Staubli VAL3: page_trajectory.pjx

--- page_trajectory.pjx ---
Parameters version=s7.8.3 stackSize=5000 millimeterUnit=true
Program file=alreadyExist.pgx
Program file=buildList.pgx
Program file=cleanUserMenu.pgx
Program file=defineTraj.pgx
Program file=deleteItem.pgx
Program file=goTo.pgx
Program file=listAdd.pgx
Program file=loadPage.pgx
Program file=main.pgx
Program file=onEnterEvent.pgx
Program file=onExit.pgx
Program file=onF1Event.pgx
Program file=onF2Event.pgx
Program file=onF3Event.pgx
Program file=onF4Event.pgx
Program file=onF5Event.pgx
Program file=onF6Event.pgx
Program file=onF7Event.pgx
Program file=onF8Event.pgx
Program file=onLeftEvent.pgx
Program file=onRightEvent.pgx
Program file=onStart.pgx
Program file=refresh.pgx
Program file=refreshDynamic.pgx
Program file=refreshStatic.pgx
Program file=selectType.pgx
Program file=showStatus.pgx
Data file=page_trajectory.dtx
Library alias=use path=Disk://public_temp/userPage/userPage.pjx
Library alias=pub path=Disk://public_temp/pub/pub.pjx
Library alias=data path=Disk://SaveData/SaveData.pjx
Library alias=cycle path=Disk://cycle/cycle.pjx

--- page_trajectory.dtx ---
num nIndex
num nKey = -1
public num nPage
num nRefresh = 2164.601
num nSelected
num nTime = 0.1
num nView
num nType
string sEvent = "hello"
string sEventImport
string sImport
public string sItems
string sList = "hello"
string sMenu[8]
  [0] = "Simulation"
  [4] = "Type"
  [5] = "Duplicate"
  [6] = "Delete"
  [7] = "New"
string sMenu8[8]
string sMenuUser[8]
string sMessage
bool bButton[8]
  [4] = true
  [5] = true
  [6] = true
  [7] = true
bool bLarge
num nIndexItem
num nOldIndex
bool bTrigger
num nClockStatus
bool bShowStatus
bool bMoveRelease
string sWorkingmode[8]
  [0] = "0 安全过度点 Joint"
  [1] = "1 Appro"
pointRx pPointTest[7]
  [0] = {fatherId=world[0]}
  [1] = {fatherId=world[0]}
  [2] = {fatherId=world[0]}
  [3] = {fatherId=world[0]}
  [4] = {fatherId=world[0]}
  [5] = {fatherId=world[0]}
  [6] = {fatherId=world[0]}
string sTrsfNum[8 6]

--- main.pgx ---
public program main()
  local bool l_bSave
  local bool l_bOverRide
  local bool l_bOk
  local bool l_bUnreached
  local string l_sMessage
begin
  //  // INIT
    call onStart()
  //  // LOOP UNTIL nKey=255
  //  nIndexItem=0
  do
    call refresh()
    nKey=getKey()
    call use:listevent(nKey,nIndex,sEvent)
    nView=use:nView
    nSelected=nIndex
		data:nPage_Traj=nIndex
    switch nKey
      case 259
        // TAB
        bLarge=!bLarge
      //  call use:setView()
      break
      case 263
        // backSpace rename
        //call onBackEvent(l_bSave)
      break
      case 32
        // space to edit Action
        //call onSpaceEvent()
      break
      case 271
        call onF1Event()
      break
      case 272
        //
        call onF2Event()
      break
      case 273
        //
        call onF3Event()
      break
      case 274
        //
        call onF4Event()
      break
      case 275
        //
        call onF5Event()
      break
      //
      case 276
        call onF6Event()
      break
      case 277
        //
        call onF7Event()
      break
      case 278
        //
        call onF8Event()
      break
      case 270
        //
        call onEnterEvent()
      break
    endSwitch
    //    endIf
    //    l_bOverRide=false
    //    // release the resource
        delay(0)
    //    if nKey==255 and isKeyPressed(289)==true
    //      call language:message(l_sMessage,143)
    //      call use:timerDialog(l_sMessage,3)
    //    endIf
    if workingMode()!=1
      call use:timerDialog("请切换成手动模式",0)
      wait(workingMode()==1)
    endIf
  until nKey==255 and isKeyPressed(289)==false
  use:bUseRefresh=true
  //  // exit
  //  call onExit(l_bSave)
end

--- alreadyExist.pgx ---
program alreadyExist(string& x_sName[], bool& x_bUndo[])
  local num l_nX
  local num l_nY
  local string l_sString
begin
//  // look if the trajectory already exist
//  l_nX=40-use:nBottomX-1
//  l_nY=use:nBottomY+1
//  call language:message(l_sString,21)
//  call use:type(l_nX,l_nY,l_sString)
//  // read the new trajectory
//  call use:read(l_nX+len(l_sString),l_nY,x_sName,10,false)
//  if !use:bUseEscape
//    call trajType:find(x_sName,x_bUndo)
//    if x_bUndo
//      call language:message(x_sName,-2)
//      popUpMsg(x_sName)
//    endIf
//  else
//    x_bUndo=true
//  endIf
end

--- buildList.pgx ---
program buildList()
  local num l_nSize
  local string l_sEvent
  local num i
  local bool l_bFound
  local num l_nCount
  local string l_sEmpty
  local num j
begin
  call use:setSizeList(0,0,38,10)
  //call use:setSizeList(15,0,18,9)
  //建立对话款
  call use:listcreate("第1槽/6槽")
  //  for i=0 to 7
  //    call use:listadd(sMenu[i])
  //  endFor
 //   call use:selectNewField(nSelected,nIndex,nView)
  for i=0 to 7
    sTrsfNum[i,0]=toString("",data:pPoinTest[i].trsf.x)
    sTrsfNum[i,1]=toString("",data:pPoinTest[i].trsf.y)
    sTrsfNum[i,2]=toString("",data:pPoinTest[i].trsf.z)
    sTrsfNum[i,3]=toString("",data:pPoinTest[i].trsf.rx)
    sTrsfNum[i,4]=toString("",data:pPoinTest[i].trsf.ry)
    sTrsfNum[i,5]=toString("",data:pPoinTest[i].trsf.rz)
  endFor

  sWorkingmode[0]="0 安全过度点 Joint"
  sWorkingmode[1]="1 Appro(摆正点，{"+sTrsfNum[1,0]+","+sTrsfNum[1,1]+","+sTrsfNum[1,2]+","+sTrsfNum[1,3]+","+sTrsfNum[1,4]+","+sTrsfNum[1,5]+"})"
  sWorkingmode[2]="2 Appro(摆正点，{"+sTrsfNum[2,0]+","+sTrsfNum[2,1]+","+sTrsfNum[2,2]+","+sTrsfNum[2,3]+","+sTrsfNum[2,4]+","+sTrsfNum[2,5]+"})"
  sWorkingmode[3]="3 Appro(到位点，{"+sTrsfNum[3,0]+","+sTrsfNum[3,1]+","+sTrsfNum[3,2]+","+sTrsfNum[3,3]+","+sTrsfNum[3,4]+","+sTrsfNum[3,5]+"})"
  sWorkingmode[4]="4 Appro(到位点，{"+sTrsfNum[4,0]+","+sTrsfNum[4,1]+","+sTrsfNum[4,2]+","+sTrsfNum[4,3]+","+sTrsfNum[4,4]+","+sTrsfNum[4,5]+"})"
  sWorkingmode[5]="5 Appro(到位点，{"+sTrsfNum[5,0]+","+sTrsfNum[5,1]+","+sTrsfNum[5,2]+","+sTrsfNum[5,3]+","+sTrsfNum[5,4]+","+sTrsfNum[5,5]+"})"
  sWorkingmode[6]="6 Appro(摆正点，{"+sTrsfNum[6,0]+","+sTrsfNum[6,1]+","+sTrsfNum[6,2]+","+sTrsfNum[6,3]+","+sTrsfNum[6,4]+","+sTrsfNum[6,5]+"})"
  sWorkingmode[7]="7 Appro(摆正点，{"+sTrsfNum[7,0]+","+sTrsfNum[7,1]+","+sTrsfNum[7,2]+","+sTrsfNum[7,3]+","+sTrsfNum[7,4]+","+sTrsfNum[7,5]+"})"

  call use:listadd(sWorkingmode)
  call use:selectNewField(nSelected,nIndex,nView)
  call use:listupdate(0)
 // nIndex=data:nPage_Traj
 // call use:selectNewField(nSelected,nIndex,nView)
end

--- cleanUserMenu.pgx ---
program cleanUserMenu()
  local num i
begin
//  // clean all the reference
//  for i=0 to size(sMenuUser)-1
//    sMenuUser[i]=""
//  endFor
end

--- defineTraj.pgx ---
program defineTraj()
  local num i
  local num l_nType
  local string l_sPath
begin
//  // select the trajectory type
//  if saveData:sTrajTypeUsing==""
//    saveData:sTrajTypeUsing=saveData:sTrajType
//  endIf
//  // search inside all the instruction
//  call saveData:getPathInstr(saveData:sTrajTypeUsing,l_sPath)
//  // check the trajType
//  if trajType:libPath()!=l_sPath and l_sPath!=""
//    i=trajType:libLoad(l_sPath)
//    delay(0)
//  endIf
//  // error
//  if i!=0
//    popUpMsg("error load traj type on ENTER"+saveData:sTrajTypeUsing+toString("",i))
//  endIf
end

--- deleteItem.pgx ---
program deleteItem(bool& x_bResult)
  local string l_sSwap
  local num l_nResult
  local string l_sMessage
  local string l_sMessage2
  local bool l_bYes
  local string l_sButton[2]
begin
//  //
//  // delete a Trajectory
//  //
//  x_bResult=false
//  // check
//  if sEvent!=""
//    l_iSwap.sType=saveData:sTrajTypeUsing
//    l_iSwap.sData=sEvent
//    call prog:findItem(l_iSwap,l_nResult,false)
//    if l_nResult==0
//      //delete it
//      call language:message(l_sMessage,81)
//      call language:getYesNo(l_sButton)
//      // ask the yes_no question
//      call use:yes_no(l_sMessage+"#"+saveData:sTrajTypeUsing+" "+sEvent,l_sButton,l_bYes)
//      x_bResult=l_bYes
//    endIf
//  endIf
end

--- goTo.pgx ---
program goTo(num x_nIndex, bool& x_bUnreached[])
  local bool l_bUnreached
  local num l_nIndexTool
  local tool l_tTool
  local num l_nSize
  local string l_sItems[2]
  local num l_nId
  local num l_nResult
begin
//  // check the cycle status
//  if !cycleStatus:bCycle and !cycleStatus:bSimulation
//    // check the working Mode
//    if cycleStatus:nWorkingMode==1 and isPowered()
//      // set the memory for the moveHold button
//      if cycleStatus:nWorkingStatus==6
//        bMoveRelease=true
//      endIf
//      // check for the index
//      if nOldIndex!=x_nIndex or (cycleStatus:nWorkingStatus!=0 and cycleStatus:nWorkingStatus!=6)
//        if !isEmpty()
//          resetMotion()
//        endIf
//        if nOldIndex!=x_nIndex
//          nOldIndex=x_nIndex
//        endIf
//      else
//        if isEmpty() and cycleStatus:nWorkingStatus==0 and bMoveRelease
//          bMoveRelease=false
//          cls()
//          // copy the item to the trajectory
//          l_sItems[0]=sEvent
//          // take the elements
//          call trajType:load(l_sItems,l_nResult)
//          call trajType:getSizeItem(false,l_nSize)
//          // MOVE
//          do
//            if x_nIndex>0
//              call use:typeMenu(7,"<<")
//            else
//              call use:typeMenu(7,"    ")
//            endIf
//            if x_nIndex<=l_nSize
//              call use:typeMenu(8,">>")
//            else
//              call use:typeMenu(8,"    ")
//            endIf
//            // get the data to move
//            call trajType:getTool(l_nIndexTool)
//            call tcp:getTool(l_tTool,l_nIndexTool)
//            call trajType:getTrajItem(l_tTraj,x_nIndex)
//            //
//            // use a sTemp mdesc to set the blend off
//            //
//            l_tTraj.nom_speed.blend=off
//            call trajType:goTo(l_tTool,l_tTraj.nom_speed,l_tTraj.moveType,x_bUnreached,x_nIndex)
//            // TO DO language
//            call use:timerDialog("Going to point: "+toString("",x_nIndex+1)+ " / "+toString("",l_nSize),0)
//            do
//              nKey=getKey()
//              call use:scroll(0,7,38,(getMoveId()-roundDown(getMoveId()))*100)
//              delay(0)
//            until isEmpty()or nKey==255 or nKey==277 or nKey==278
//            // continue
//            if isEmpty() or (nKey==278 and x_nIndex<l_nSize)
//              if isEmpty()
//                call use:timerDialog("At point: "+toString("",x_nIndex+1)+ " / "+toString("",l_nSize),1)
//              endIf
//              x_nIndex=x_nIndex+1
//            elseIf nKey==277 and x_nIndex>0
//              // decrease
//              x_nIndex=x_nIndex-1
//            else
//              delay(1)
//            endIf
//            // release
//            resetMotion()
//          until x_bUnreached or nKey==255 or x_nIndex>=l_nSize or(x_nIndex==l_nSize and l_nSize==1)
//          // refresh
//          use:bUseRefresh=true
//        endIf
//      endIf
//    else
//      // reset the cycle
//      if cycleStatus:nWorkingMode!=1 or !isPowered()
//        resetMotion()
//      endIf
//    endIf
//  endIf
end

--- loadPage.pgx ---
program loadPage(string x_sPage, string& x_sItems[])
// load the next page
  local num i
  local string l_sMessage
begin
//  // look if the page libload is correct
//  i=page:libLoad(x_sPage)
//  delay(0)
//  if i!=0
//    logMsg("[KERNEL] INTERFACE:PAGE LIBLOAD "+x_sPage+" result "+toString("",i))
//    call language:message(l_sMessage,-7)
//    popUpMsg(l_sMessage+x_sPage+" ; "+toString("",i))
//  else
//    // copy all the field from x_sItems to the next page
//    call use:stringCopy(x_sItems,page:sItems)
//    call page:main()
//  endIf
end

--- onExit.pgx ---
program onExit(bool x_bSave)
  local string l_sEmpty
  local num l_nResult
  local string l_sMessage
begin
//  // resetMotion
//  if !cycleStatus:bCycle
//    resetMotion()
//  endIf
//  if x_bSave
//    l_sEmpty=""
//    l_nResult=0
//    call trajType:onSave(l_sEmpty)
//    // show the message
//    call language:message(l_sMessage,-4)
//    call use:timerDialog(l_sMessage,1)
//  endIf
end

--- onF1Event.pgx ---
program onF1Event()
  local bool l_bYes
  local string l_sMessage
  local string l_sItem
  local num l_nResult
begin
//  // look if the bButton is enable
//  if bButton[0]
//    //
//    //SIMULATION
//    //
//    if !cycleStatus:bCycle and sEvent!=""
//      // load the production page
//      call loadPage("Disk://trajectory/page_simulation",sEvent)
//      // save the moveHold
//      bMoveRelease=false
//    endIf
//  endIf
end

--- onF2Event.pgx ---
program onF2Event()
  local string l_sMessage
  local string l_sEvent
  local string l_sFilter
  local num l_nIndex
  local num i
begin
//  // look if the bButton is enable
//  if bButton[1]
//    //
//    // make a selection list
//    //
//    // 0) Filter by name
//    //
//    call use:clear(0,13)
//    call use:type(5,13,sMenu[1])
//    call language:message(l_sMessage,85)
//    call use:timerDialog(l_sMessage+": ",0)
//    l_sFilter=saveData:sTrajFilter
//    call use:read(20+(len(l_sMessage)/2)+1,5,l_sFilter,10,false)
//    if !use:bUseEscape
//      saveData:sTrajFilter=l_sFilter
//    endIf

//    // update
//    call buildList()
//    use:bUseRefresh=true
//    // release the key
//    call use:nullKey(nKey)
//  endIf
end

--- onF3Event.pgx ---
program onF3Event()
begin
//  // look if the bButton is enable
//  if bButton[2]
//    //
//  endIf
end

--- onF4Event.pgx ---
program onF4Event()
  local string l_sMessage
  local bool l_bImport
  local string l_sPath[2]
  local num l_nLocal
  local num l_nKey
  local bool l_bDone
  local num l_nOldValue[4]
  local num i
  local num l_nDefault
  local string l_sButton[2]
  local string l_sItem
begin
//  // look if the bButton is enable
//  if bButton[3]
//    //
//  endIf
end

--- onF8Event.pgx ---
program onF8Event()
  local string l_sNew
  local bool l_bUndo
  local num l_nResult
begin
//  // look if the bButton is enable
  if bButton[7]
    call cycle:wizard()
    call buildList()
  endIf
end

--- onLeftEvent.pgx ---
program onLeftEvent(bool& x_bSave)
  local num i
  local num l_nType
  local string l_sPath
  local string l_sEmpty
  local num l_nResult
  local string l_sMessage
begin
//  // left click
//  //
//  //
//  // select the previous one
//  //
//  if x_bSave
//    x_bSave=false
//    l_sEmpty=""
//    l_nResult=0
//    call trajType:onSave(l_sEmpty)
//    // show the message
//    call language:message(l_sMessage,-4)
//    call use:timerDialog(l_sMessage,1)
//  endIf
//  // check it
//  do
//    nType=(nType+size(saveData:sTrajType)-1)%(size(saveData:sTrajType))
//    saveData:sTrajTypeUsing=saveData:sTrajType[nType]
//    if saveData:sTrajType[nType]!=""
//      // find the good id
//      call saveData:getPathInstr(saveData:sTrajType[nType],l_sPath)
//    endIf
//  until saveData:sTrajType[nType]!=""
//  // load the type
//  if trajType:libPath()!=l_sPath and l_sPath!=""
//    i=trajType:libLoad(l_sPath)
//    delay(0)
//  endIf
//  if l_sPath==""
//    popUpMsg("error load traj type on ENTER "+saveData:sTrajTypeUsing+toString("",i))
//  endIf
//  // clean the user MENU
//  call cleanUserMenu()
//  // rebuild the list
//  call buildList()
end

--- onStart.pgx ---
program onStart()
  local num i
begin
  cls()
  userPage()
  call use:nullKey(nKey)
  call buildList()
  call refreshStatic()
end

--- refresh.pgx ---
program refresh()
// // page refresh
begin
    if  (nKey>=270 and nKey<=278) or use:bUseRefresh==true
    cls()
    call refreshStatic()
    call buildList()
    call refreshDynamic()
    if abs(clock()-nRefresh)>nTime
      call refreshDynamic()
    endIf
  endIf
end

--- refreshDynamic.pgx ---
program refreshDynamic()
  local string l_sMessage
begin
//  // DO NOT CHANGE
  nRefresh=clock()
  use:bUseRefresh=false
//  //
//  // ADD HERE
//  //
end

--- refreshStatic.pgx ---
program refreshStatic()
  local string l_sMessage
  local num i
  local string l_sMenu
begin
  title("编辑-1号石墨舟A面方片")
  l_sMenu=",,,,,吸片,放片,向导"
  // define the menu
  call use:stringToArray(l_sMenu,sMenu)
  call use:typeMenu(6,"吸片")
  call use:typeMenu(7,"放片")
  call use:typeMenu(8,"向导")
  // set the menu
  //call use:setMenu(sMenu,true,2)
  //call use:getMenu(sMenu,bButton)
  //  cls()
  //  //
  //  // set the view of the page..
  //  //
  //  // SET THE PAGE NUMBER
  //  use:nPage=1010
  //  // USE <>PROFILE for <>PAGE
  //  use:nPage=use:nPage+abs(limit(saveData:mode,0,2)-2)
  //  if cycleStatus:bCycle
  //    use:nPage=use:nPage+3
  //  endIf
  //  // load the menu page
  //  if saveData:language!="japanese"
  //    // SET THE VIEW OF THE PAGE
  //    call language:page(l_sMessage,use:nPage)
  //    // define the menu
  //    call use:stringToArray(l_sMessage,sMenu)
  //  else
  //    // japanese use the array for the menu
  //    call language:page(sMenu8,use:nPage)
  //    call use:stringCopy(sMenu8,sMenu)
  //  endIf
  //  //
  //  // polymorphism
  //  //
  //  // get the user Menu or special one
  //  call trajType:getFunctionSel(sMenuUser)
  //  // OVERRIDE
  //  for i=0 to size(sMenuUser)-1
  //    if sMenuUser[i]!=""
  //      sMenu[i]=sMenuUser[i]
  //    endIf
  //  endFor
  //  // set the menu
  //  if saveData:language!="japanese"
  //    call use:setMenu(sMenu,true,3)
  //  else
  //    call use:setMenu(sMenu,false,3)
  //  endIf
  //  call use:getMenu(sMenu,bButton)
  //  //
  //  // CREATE THE LIST
  //  //
  //  // define your list size for default
  //  call use:setSizeList(19,0,19,11)
  //  call use:setView(bLarge)
  //  //
  //  call use:listcreate(saveData:sTrajTypeUsing)
  //  //
  //  call use:listadd(sList)
  //  //
  //  // refresh the list
  //  call use:selectNewField(nSelected,nIndex,nView)
  //  //
  //  // is a filter using ??
  //  if  saveData:sTrajFilter!=""
  //    call language:message(l_sMessage,64)
  //    call use:type(0,1,l_sMessage+">"+saveData:sTrajFilter)
  //  else
  //    // clean
  //    call use:typeLen(0,1," ",use:nBottomX)
  //  endIf
end

--- showStatus.pgx ---
program showStatus()
  local joint l_jHere
  local point l_pHere
  local string l_sMessage[2]
  local tool l_tTool
  local num l_nIndexTool
begin
//  //
//  // show an dialog box with
//  // the current Joint/cartesian position
//  //
//  call trajType:getTool(l_nIndexTool)
//  call tcp:getTool(l_tTool,l_nIndexTool)
//  if cycleStatus:nWorkingStatus>1 and cycleStatus:nWorkingStatus<5 and cycleStatus:nWorkingMode==1
//    // set a timer of x second then the message disappear ..
//    if !bTrigger
//      nClockStatus=clock()
//      bTrigger=true
//      bShowStatus=true
//    endIf
//    if clock()-nClockStatus<saveData:nTimeDialog
//      if cycleStatus:nWorkingStatus==2
//        l_jHere=herej()
//        l_sMessage="J1:"+toString("7.1",l_jHere.j1)
//        l_sMessage=l_sMessage+"  J2:"+toString("7.1",l_jHere.j2)+"#"
//        l_sMessage=l_sMessage+"J3:"+toString("7.1",l_jHere.j3)
//        l_sMessage=l_sMessage+"  J4:"+toString("7.1",l_jHere.j4)
//        //l_sMessage=l_sMessage+"  J5:"+toString("7.1",l_jHere.j5)
//        //l_sMessage=l_sMessage+"  J6:"+toString("7.1",l_jHere.j6)
//      else
//        l_pHere=here(l_tTool,saveData:fFrameItem[saveData:nFrameActive].fFrame)
//        l_sMessage="X :"+toString("7.1",l_pHere.trsf.x)
//        l_sMessage=l_sMessage+"  Y :"+toString("7.1",l_pHere.trsf.y)
//        l_sMessage=l_sMessage+"  Z :"+toString("7.1",l_pHere.trsf.z)+"#"
//        l_sMessage=l_sMessage+"RX:"+toString("7.1",l_pHere.trsf.rx)
//        l_sMessage=l_sMessage+"  RY:"+toString("7.1",l_pHere.trsf.ry)
//        l_sMessage=l_sMessage+"  RZ:"+toString("7.1",l_pHere.trsf.rz)
//      endIf
//      call use:timerDialog(l_sMessage,0)
//    else
//      // disable it
//      bShowStatus=false
//    endIf
//  else
//    // reset it
//    if bTrigger and !cycleStatus:bCycle
//      resetMotion()
//    endIf
//    bTrigger=false
//    bShowStatus=false
//  endIf
end
